FUNCTION_BLOCK BLINK
VAR_INPUT
	OnTime : TIME;
    OffTime : TIME;
END_VAR

VAR_OUTPUT
    OUT : BOOL;
END_VAR

VAR
    fbTon  : TON;
    fbToff : TON;
END_VAR

fbTon.PT  := OnTime;
fbToff.PT := OffTime;

fbTon.IN := NOT fbToff.Q;
fbTon();

fbToff.IN := fbTon.Q;
fbToff();

Out := fbTon.Q;

END_FUNCTION_BLOCK

(* stored: Version 1.1.0.1
   POU BLINK: Id {dd599460-7c02-412a-aaaa-8ca0d00c32a3}, SpecialFunc None *)
